TEXTLIST ScreenNames
  801 = 'EtherCAT Diagnostics' | 汉语: '汉语'
  802 = 'PROFIBUS Diagnostics' | 汉语: '汉语'
  803 = 'PROFINET Diagnostics' | 汉语: '汉语'
  800 = 'I/O Memory Display'
  40 = 'Machine Layout'
  30 = 'Menu Screen 1'
  31 = 'Menu Screen 2'
  32 = 'Menu Screen 3'
  20 = 'Alarms'
  21 = 'Alarm View'
  1 = 'Mode Screen'
  10 = 'Motions'
  500 = 'Part Screen'
  900 = 'About'
  901 = 'HMI Screen'
  401 = 'Machine Units'
  402 = 'Axis Screen'
  403 = 'Language Screen'
  32767 = 'No Screen Detected'
  501 = 'Cycle Time'
  11 = 'Axis Data'
  700 = 'Safety Status'
  701 = 'Safety Checksum'
  2 = 'Mode Screen Rows'
   = ''
END_TEXTLIST

(* stored: Version 1.1.0.1, ProductVersion 3.1.4024.12
   TextList ScreenNames: Id {45969ee7-d1fd-4f73-bec4-132b70f9ad88} *)
